PROGRAM MAIN
VAR
	root 		: Directory('root');
	
	archive1	: Archive('archivo1.txt', 10);			    
    archive2  	: Archive('archivo2.txt', 30);
    archive3 	: Archive('archivo3.txt', 120);
    archive4 	: Archive('archivo4.txt', 800);
    archive5 	: Archive('archivo5.txt', 340);

    archive6 	: Archive('archivo6.txt', 122);
    archive7 	: Archive('archivo7.txt', 391);

    dir1 		: Directory('dir1');
    dir2 		: Directory('dir2');
    dir3 		: Directory('dir3');

	bExecute	: BOOL;	
	sMsg 		: STRING;

END_VAR

IF bExecute THEN
	
	bExecute := FALSE;
	
	dir1.ResetSize();
	dir2.ResetSize();
	dir3.ResetSize();
	root.ResetSize();
 
	dir1.AddChild(archive1); // 10
 	dir1.AddChild(archive6); // 122
 	dir2.AddChild(archive2); // 30
 	dir3.AddChild(archive3); // 120
 	dir3.AddChild(archive4); // 800
 	dir1.AddChild(dir3); // 120+800

 	root.AddChild(dir1); // dir1 = 120+800+10+122 = 1052
 	root.AddChild(dir2); // dir2 = 30
 	root.AddChild(archive5); // 340
 	root.AddChild(archive7); // 391
	
	// root = 1052+30+340+391 = 1813
	sMsg := CONCAT(STR1:= root.Name , STR2:= CONCAT(STR1:= ' is: ' , STR2:= TO_STRING(root.GetSize) ) );
	ADSLOGSTR(msgCtrlMask:= ADSLOG_MSGTYPE_LOG, msgFmtStr:= 'The size of the directory %s ' , strArg:= sMsg);
	
	// dir1 = 10+122+120+800 = 1052
	sMsg := CONCAT(STR1:= dir1.Name , STR2:= CONCAT(STR1:= ' is: ' , STR2:= TO_STRING(dir1.GetSize) ) );
	ADSLOGSTR(msgCtrlMask:= ADSLOG_MSGTYPE_LOG, msgFmtStr:= 'The size of the directory %s ' , strArg:= sMsg);
	
	// dir2 = 30
	sMsg := CONCAT(STR1:= dir2.Name , STR2:= CONCAT(STR1:= ' is: ' , STR2:= TO_STRING(dir2.GetSize) ) );
	ADSLOGSTR(msgCtrlMask:= ADSLOG_MSGTYPE_LOG, msgFmtStr:= 'The size of the directory %s ' , strArg:= sMsg);
	
	// dir3 = 120+800 = 922
	sMsg := CONCAT(STR1:= dir3.Name , STR2:= CONCAT(STR1:= ' is: ' , STR2:= TO_STRING(dir3.GetSize) ) );
	ADSLOGSTR(msgCtrlMask:= ADSLOG_MSGTYPE_LOG, msgFmtStr:= 'The size of the directory %s ' , strArg:= sMsg);	
	
END_IF

END_PROGRAM

(* stored: Version 1.1.0.1, ProductVersion 3.1.4024.12
   POU MAIN: Id {3d6c1cda-8968-4d01-8af4-51ef2b43d90c}, SpecialFunc None *)
